FUNCTION_BLOCK testttt
VAR_INPUT
END_VAR
VAR_OUTPUT
END_VAR
VAR
END_VAR

END_FUNCTION_BLOCK

(* stored: Version 1.1.0.1, ProductVersion 3.1.4026.12
   POU testttt: Id {d6330784-6436-4763-96b2-1a100faf9b8c}, SpecialFunc None *)
